PROGRAM MAIN
VAR
	rParam: I_Object;

	_init: BOOL;
END_VAR

IF NOT _init THEN
	
	F_Change_Param(
		G.A1.Get_Child('B1').Get_Child('tB'),
		'TRUE');
		
	rParam := G.A1.Get_Child('C1').Get_Child('tR');
	F_Change_Param(rParam, '0.7');

	
	_init := TRUE;
END_IF

END_PROGRAM

(* stored: Version 1.1.0.1, ProductVersion 3.1.4024.12
   POU MAIN: Id {e6bb2c3e-4cb9-4dca-9990-7f3dc31798cf}, SpecialFunc None *)
